// TIA Portal V19 export
FUNCTION "SUGAR TRANSFER CYCLE" : Void   // FC26, LAD
{ S7_Optimized_Access := 'TRUE' }
// stored: SetENOAutomatically false
   VAR_TEMP   // added for the SCL form of the ladder/FBD networks
      _w1 : Bool;
   END_VAR
BEGIN

REGION Network 1: TRANSFER SELECT
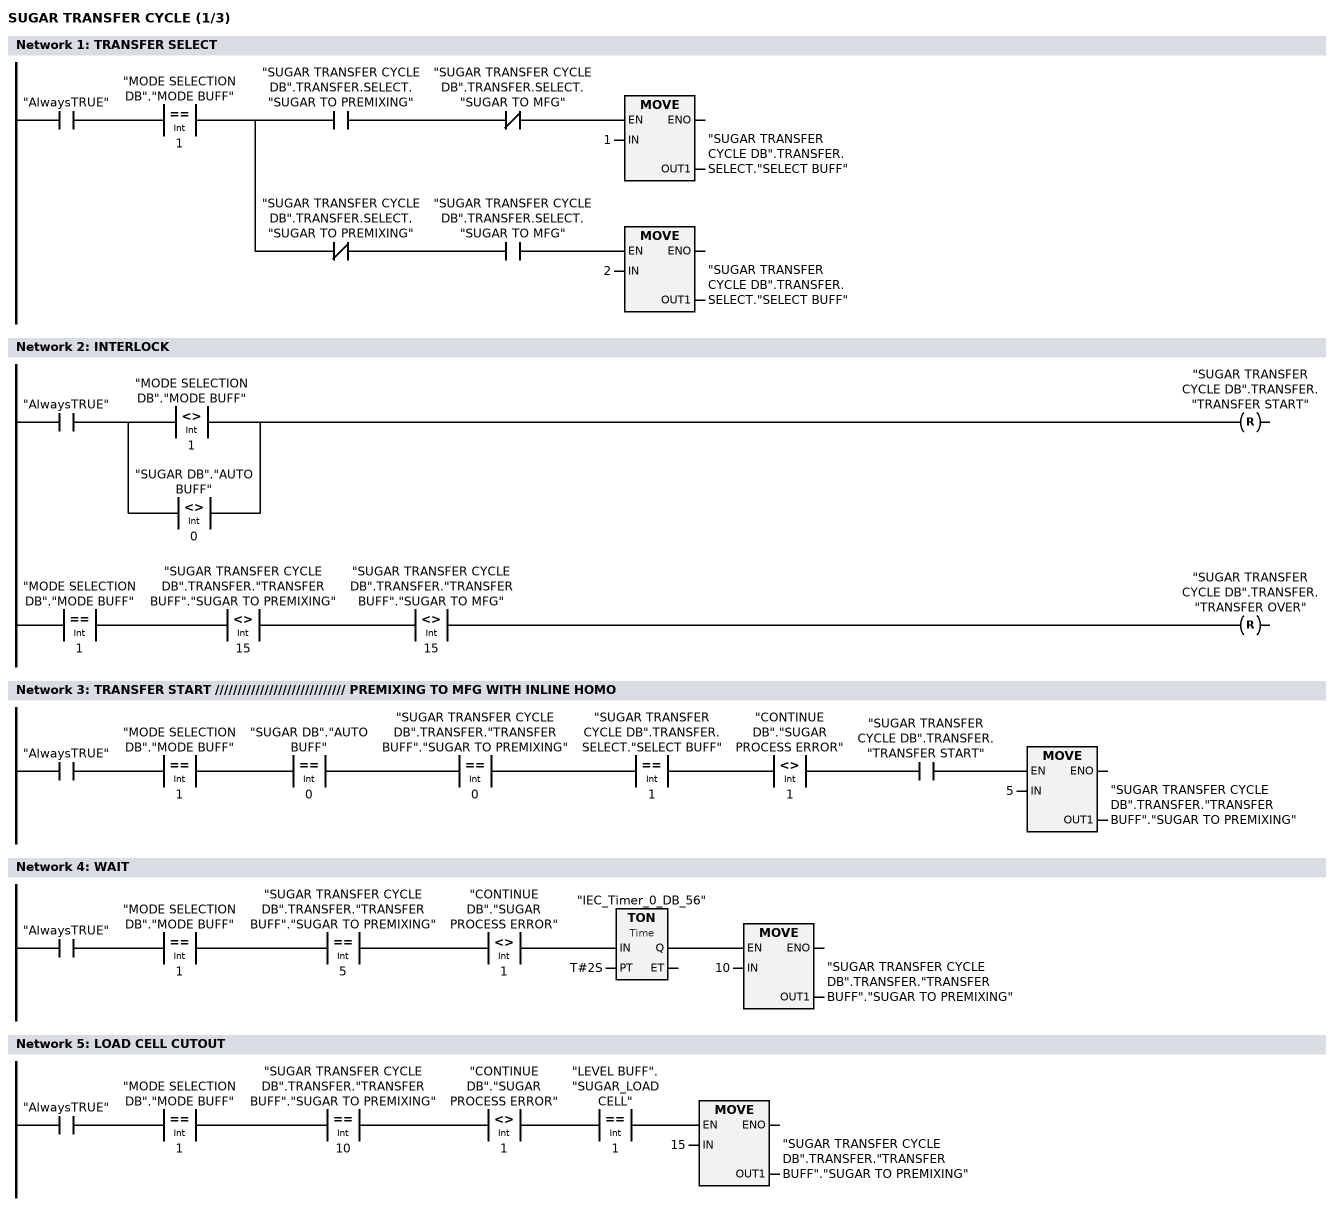
   RUNG wire#powerrail
      Contact( "AlwaysTRUE" )
      { S7_Templates := "SrcType := Int" } EQ_Contact(in1 := "MODE SELECTION DB"."MODE BUFF", in2 := 1)
      wire#w1
      Contact( "SUGAR TRANSFER CYCLE DB".TRANSFER.SELECT."SUGAR TO PREMIXING" )
      I_Contact( "SUGAR TRANSFER CYCLE DB".TRANSFER.SELECT."SUGAR TO MFG" )
      Move(in := 1, out1 => "SUGAR TRANSFER CYCLE DB".TRANSFER.SELECT."SELECT BUFF")
   END_RUNG
   RUNG wire#w1
      I_Contact( "SUGAR TRANSFER CYCLE DB".TRANSFER.SELECT."SUGAR TO PREMIXING" )
      Contact( "SUGAR TRANSFER CYCLE DB".TRANSFER.SELECT."SUGAR TO MFG" )
      Move(in := 2, out1 => "SUGAR TRANSFER CYCLE DB".TRANSFER.SELECT."SELECT BUFF")
   END_RUNG
   // the same network as SCL:
   #_w1 := "AlwaysTRUE" AND ("MODE SELECTION DB"."MODE BUFF" = 1);
   IF #_w1 AND "SUGAR TRANSFER CYCLE DB".TRANSFER.SELECT."SUGAR TO PREMIXING" AND NOT "SUGAR TRANSFER CYCLE DB".TRANSFER.SELECT."SUGAR TO MFG" THEN
       "SUGAR TRANSFER CYCLE DB".TRANSFER.SELECT."SELECT BUFF" := 1;
   END_IF;
   IF #_w1 AND NOT "SUGAR TRANSFER CYCLE DB".TRANSFER.SELECT."SUGAR TO PREMIXING" AND "SUGAR TRANSFER CYCLE DB".TRANSFER.SELECT."SUGAR TO MFG" THEN
       "SUGAR TRANSFER CYCLE DB".TRANSFER.SELECT."SELECT BUFF" := 2;
   END_IF;
END_REGION

REGION Network 2: INTERLOCK
   RUNG wire#powerrail
      Contact( "AlwaysTRUE" )
      wire#w1
      { S7_Templates := "SrcType := Int" } NE_Contact(in1 := "MODE SELECTION DB"."MODE BUFF", in2 := 1)
      wire#w2
      R_Coil( "SUGAR TRANSFER CYCLE DB".TRANSFER."TRANSFER START" )
   END_RUNG
   RUNG wire#w1
      { S7_Templates := "SrcType := Int" } NE_Contact(in1 := "SUGAR DB"."AUTO BUFF", in2 := 0)
   END_RUNG wire#w2
   RUNG wire#powerrail
      { S7_Templates := "SrcType := Int" } EQ_Contact(in1 := "MODE SELECTION DB"."MODE BUFF", in2 := 1)
      { S7_Templates := "SrcType := Int" } NE_Contact(in1 := "SUGAR TRANSFER CYCLE DB".TRANSFER."TRANSFER BUFF"."SUGAR TO PREMIXING", in2 := 15)
      { S7_Templates := "SrcType := Int" } NE_Contact(in1 := "SUGAR TRANSFER CYCLE DB".TRANSFER."TRANSFER BUFF"."SUGAR TO MFG", in2 := 15)
      R_Coil( "SUGAR TRANSFER CYCLE DB".TRANSFER."TRANSFER OVER" )
   END_RUNG
   // the same network as SCL:
   IF "AlwaysTRUE" AND (("MODE SELECTION DB"."MODE BUFF" <> 1) OR ("SUGAR DB"."AUTO BUFF" <> 0)) THEN
       "SUGAR TRANSFER CYCLE DB".TRANSFER."TRANSFER START" := FALSE;
   END_IF;
   IF ("MODE SELECTION DB"."MODE BUFF" = 1) AND ("SUGAR TRANSFER CYCLE DB".TRANSFER."TRANSFER BUFF"."SUGAR TO PREMIXING" <> 15) AND ("SUGAR TRANSFER CYCLE DB".TRANSFER."TRANSFER BUFF"."SUGAR TO MFG" <> 15) THEN
       "SUGAR TRANSFER CYCLE DB".TRANSFER."TRANSFER OVER" := FALSE;
   END_IF;
END_REGION

REGION Network 3: TRANSFER START ///////////////////////////// PREMIXING TO MFG WITH INLINE HOMO
   RUNG wire#powerrail
      Contact( "AlwaysTRUE" )
      { S7_Templates := "SrcType := Int" } EQ_Contact(in1 := "MODE SELECTION DB"."MODE BUFF", in2 := 1)
      { S7_Templates := "SrcType := Int" } EQ_Contact(in1 := "SUGAR DB"."AUTO BUFF", in2 := 0)
      { S7_Templates := "SrcType := Int" } EQ_Contact(in1 := "SUGAR TRANSFER CYCLE DB".TRANSFER."TRANSFER BUFF"."SUGAR TO PREMIXING", in2 := 0)
      { S7_Templates := "SrcType := Int" } EQ_Contact(in1 := "SUGAR TRANSFER CYCLE DB".TRANSFER.SELECT."SELECT BUFF", in2 := 1)
      { S7_Templates := "SrcType := Int" } NE_Contact(in1 := "CONTINUE DB"."SUGAR PROCESS ERROR", in2 := 1)
      Contact( "SUGAR TRANSFER CYCLE DB".TRANSFER."TRANSFER START" )
      Move(in := 5, out1 => "SUGAR TRANSFER CYCLE DB".TRANSFER."TRANSFER BUFF"."SUGAR TO PREMIXING")
   END_RUNG
   // the same network as SCL:
   IF "AlwaysTRUE" AND ("MODE SELECTION DB"."MODE BUFF" = 1) AND ("SUGAR DB"."AUTO BUFF" = 0) AND ("SUGAR TRANSFER CYCLE DB".TRANSFER."TRANSFER BUFF"."SUGAR TO PREMIXING" = 0) AND ("SUGAR TRANSFER CYCLE DB".TRANSFER.SELECT."SELECT BUFF" = 1) AND ("CONTINUE DB"."SUGAR PROCESS ERROR" <> 1) AND "SUGAR TRANSFER CYCLE DB".TRANSFER."TRANSFER START" THEN
       "SUGAR TRANSFER CYCLE DB".TRANSFER."TRANSFER BUFF"."SUGAR TO PREMIXING" := 5;
   END_IF;
END_REGION

REGION Network 4: WAIT
   RUNG wire#powerrail
      Contact( "AlwaysTRUE" )
      { S7_Templates := "SrcType := Int" } EQ_Contact(in1 := "MODE SELECTION DB"."MODE BUFF", in2 := 1)
      { S7_Templates := "SrcType := Int" } EQ_Contact(in1 := "SUGAR TRANSFER CYCLE DB".TRANSFER."TRANSFER BUFF"."SUGAR TO PREMIXING", in2 := 5)
      { S7_Templates := "SrcType := Int" } NE_Contact(in1 := "CONTINUE DB"."SUGAR PROCESS ERROR", in2 := 1)
      { S7_Templates := "time_type := Time" } "IEC_Timer_0_DB_56".TON(pt := T#2S, et =>)
      Move(in := 10, out1 => "SUGAR TRANSFER CYCLE DB".TRANSFER."TRANSFER BUFF"."SUGAR TO PREMIXING")
   END_RUNG
   // the same network as SCL:
   "IEC_Timer_0_DB_56".TON(IN := "AlwaysTRUE" AND ("MODE SELECTION DB"."MODE BUFF" = 1) AND ("SUGAR TRANSFER CYCLE DB".TRANSFER."TRANSFER BUFF"."SUGAR TO PREMIXING" = 5) AND ("CONTINUE DB"."SUGAR PROCESS ERROR" <> 1),
                           PT := T#2S);
   IF "IEC_Timer_0_DB_56".Q THEN
       "SUGAR TRANSFER CYCLE DB".TRANSFER."TRANSFER BUFF"."SUGAR TO PREMIXING" := 10;
   END_IF;
END_REGION

REGION Network 5: LOAD CELL CUTOUT
   RUNG wire#powerrail
      Contact( "AlwaysTRUE" )
      { S7_Templates := "SrcType := Int" } EQ_Contact(in1 := "MODE SELECTION DB"."MODE BUFF", in2 := 1)
      { S7_Templates := "SrcType := Int" } EQ_Contact(in1 := "SUGAR TRANSFER CYCLE DB".TRANSFER."TRANSFER BUFF"."SUGAR TO PREMIXING", in2 := 10)
      { S7_Templates := "SrcType := Int" } NE_Contact(in1 := "CONTINUE DB"."SUGAR PROCESS ERROR", in2 := 1)
      { S7_Templates := "SrcType := Int" } EQ_Contact(in1 := "LEVEL BUFF"."SUGAR_LOAD CELL", in2 := 1)
      Move(in := 15, out1 => "SUGAR TRANSFER CYCLE DB".TRANSFER."TRANSFER BUFF"."SUGAR TO PREMIXING")
   END_RUNG
   // the same network as SCL:
   IF "AlwaysTRUE" AND ("MODE SELECTION DB"."MODE BUFF" = 1) AND ("SUGAR TRANSFER CYCLE DB".TRANSFER."TRANSFER BUFF"."SUGAR TO PREMIXING" = 10) AND ("CONTINUE DB"."SUGAR PROCESS ERROR" <> 1) AND ("LEVEL BUFF"."SUGAR_LOAD CELL" = 1) THEN
       "SUGAR TRANSFER CYCLE DB".TRANSFER."TRANSFER BUFF"."SUGAR TO PREMIXING" := 15;
   END_IF;
END_REGION

REGION Network 6: TIMER
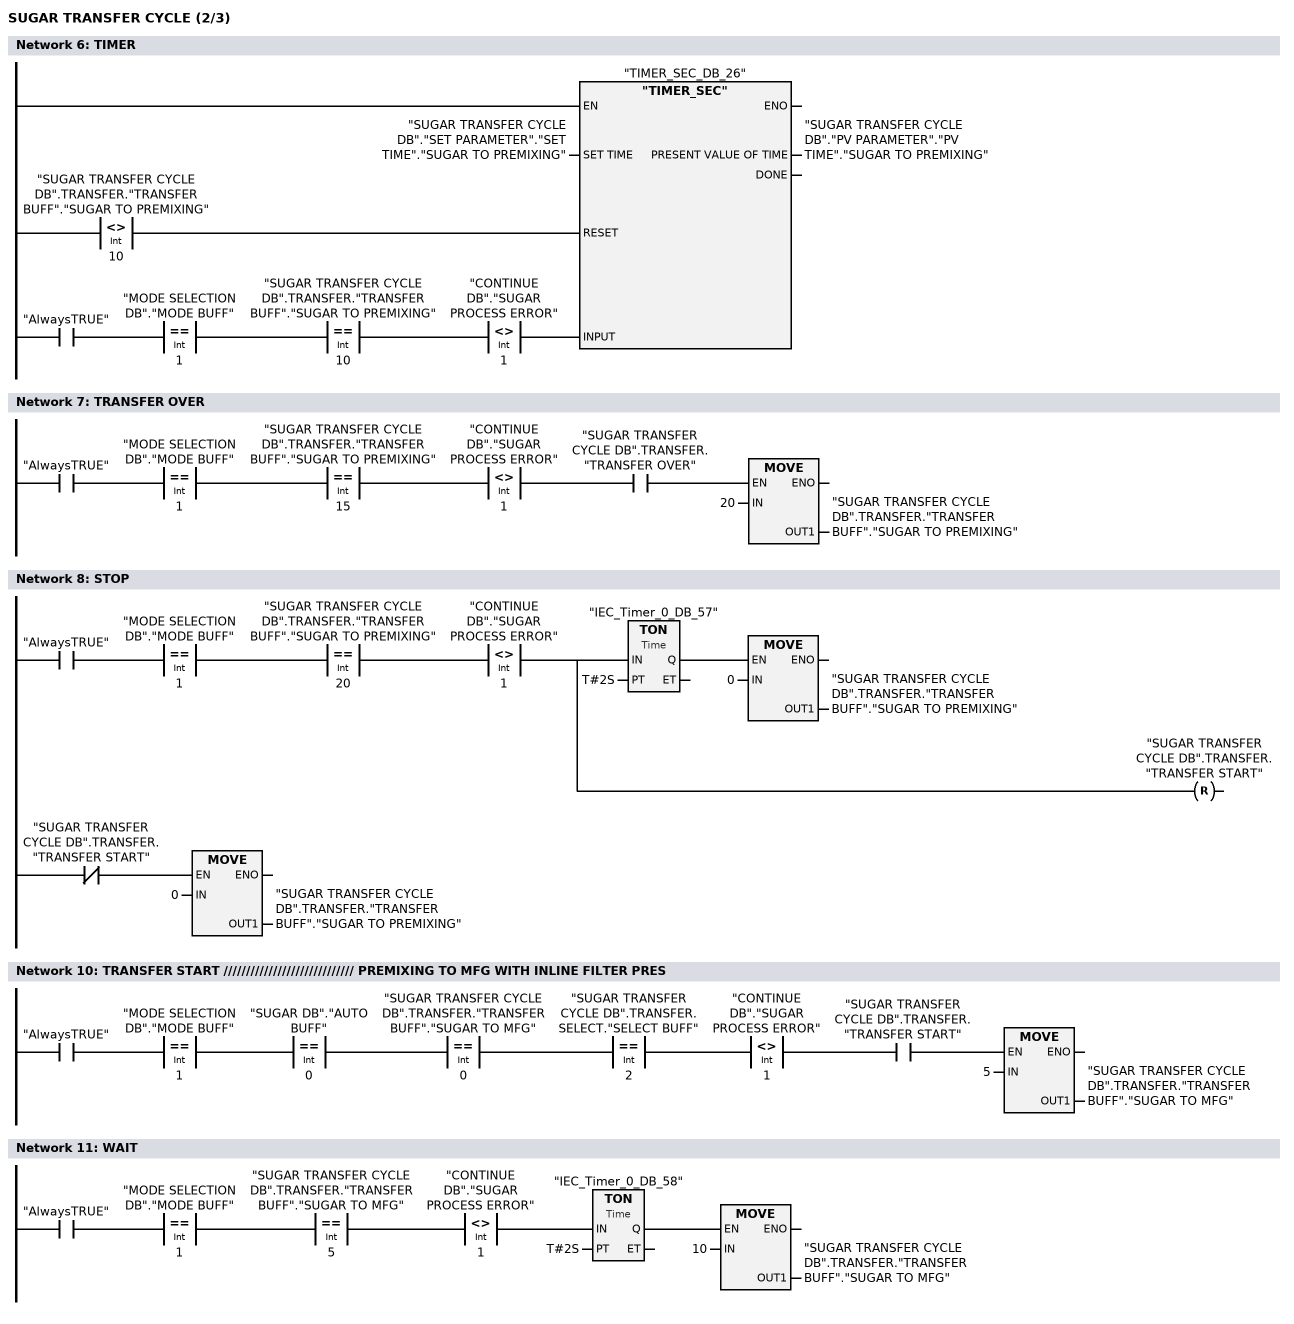
   RUNG wire#powerrail
      "TIMER_SEC_DB_26"(RESET := wire#w1, INPUT := wire#w2, "SET TIME" := "SUGAR TRANSFER CYCLE DB"."SET PARAMETER"."SET TIME"."SUGAR TO PREMIXING", "PRESENT VALUE OF TIME" => "SUGAR TRANSFER CYCLE DB"."PV PARAMETER"."PV TIME"."SUGAR TO PREMIXING", DONE =>)
   END_RUNG
   RUNG wire#powerrail
      { S7_Templates := "SrcType := Int" } NE_Contact(in1 := "SUGAR TRANSFER CYCLE DB".TRANSFER."TRANSFER BUFF"."SUGAR TO PREMIXING", in2 := 10)
   END_RUNG wire#w1
   RUNG wire#powerrail
      Contact( "AlwaysTRUE" )
      { S7_Templates := "SrcType := Int" } EQ_Contact(in1 := "MODE SELECTION DB"."MODE BUFF", in2 := 1)
      { S7_Templates := "SrcType := Int" } EQ_Contact(in1 := "SUGAR TRANSFER CYCLE DB".TRANSFER."TRANSFER BUFF"."SUGAR TO PREMIXING", in2 := 10)
      { S7_Templates := "SrcType := Int" } NE_Contact(in1 := "CONTINUE DB"."SUGAR PROCESS ERROR", in2 := 1)
   END_RUNG wire#w2
   // the same network as SCL:
   "TIMER_SEC_DB_26"("SET TIME" := "SUGAR TRANSFER CYCLE DB"."SET PARAMETER"."SET TIME"."SUGAR TO PREMIXING",   // "TIMER_SEC"
                     RESET := "SUGAR TRANSFER CYCLE DB".TRANSFER."TRANSFER BUFF"."SUGAR TO PREMIXING" <> 10,
                     INPUT := "AlwaysTRUE" AND ("MODE SELECTION DB"."MODE BUFF" = 1) AND ("SUGAR TRANSFER CYCLE DB".TRANSFER."TRANSFER BUFF"."SUGAR TO PREMIXING" = 10) AND ("CONTINUE DB"."SUGAR PROCESS ERROR" <> 1),
                     "PRESENT VALUE OF TIME" => "SUGAR TRANSFER CYCLE DB"."PV PARAMETER"."PV TIME"."SUGAR TO PREMIXING");
END_REGION

REGION Network 7: TRANSFER OVER
   RUNG wire#powerrail
      Contact( "AlwaysTRUE" )
      { S7_Templates := "SrcType := Int" } EQ_Contact(in1 := "MODE SELECTION DB"."MODE BUFF", in2 := 1)
      { S7_Templates := "SrcType := Int" } EQ_Contact(in1 := "SUGAR TRANSFER CYCLE DB".TRANSFER."TRANSFER BUFF"."SUGAR TO PREMIXING", in2 := 15)
      { S7_Templates := "SrcType := Int" } NE_Contact(in1 := "CONTINUE DB"."SUGAR PROCESS ERROR", in2 := 1)
      Contact( "SUGAR TRANSFER CYCLE DB".TRANSFER."TRANSFER OVER" )
      Move(in := 20, out1 => "SUGAR TRANSFER CYCLE DB".TRANSFER."TRANSFER BUFF"."SUGAR TO PREMIXING")
   END_RUNG
   // the same network as SCL:
   IF "AlwaysTRUE" AND ("MODE SELECTION DB"."MODE BUFF" = 1) AND ("SUGAR TRANSFER CYCLE DB".TRANSFER."TRANSFER BUFF"."SUGAR TO PREMIXING" = 15) AND ("CONTINUE DB"."SUGAR PROCESS ERROR" <> 1) AND "SUGAR TRANSFER CYCLE DB".TRANSFER."TRANSFER OVER" THEN
       "SUGAR TRANSFER CYCLE DB".TRANSFER."TRANSFER BUFF"."SUGAR TO PREMIXING" := 20;
   END_IF;
END_REGION

REGION Network 8: STOP
   RUNG wire#powerrail
      Contact( "AlwaysTRUE" )
      { S7_Templates := "SrcType := Int" } EQ_Contact(in1 := "MODE SELECTION DB"."MODE BUFF", in2 := 1)
      { S7_Templates := "SrcType := Int" } EQ_Contact(in1 := "SUGAR TRANSFER CYCLE DB".TRANSFER."TRANSFER BUFF"."SUGAR TO PREMIXING", in2 := 20)
      { S7_Templates := "SrcType := Int" } NE_Contact(in1 := "CONTINUE DB"."SUGAR PROCESS ERROR", in2 := 1)
      wire#w1
      { S7_Templates := "time_type := Time" } "IEC_Timer_0_DB_57".TON(pt := T#2S, et =>)
      Move(in := 0, out1 => "SUGAR TRANSFER CYCLE DB".TRANSFER."TRANSFER BUFF"."SUGAR TO PREMIXING")
   END_RUNG
   RUNG wire#w1
      R_Coil( "SUGAR TRANSFER CYCLE DB".TRANSFER."TRANSFER START" )
   END_RUNG
   RUNG wire#powerrail
      I_Contact( "SUGAR TRANSFER CYCLE DB".TRANSFER."TRANSFER START" )
      Move(in := 0, out1 => "SUGAR TRANSFER CYCLE DB".TRANSFER."TRANSFER BUFF"."SUGAR TO PREMIXING")
   END_RUNG
   // the same network as SCL:
   #_w1 := "AlwaysTRUE" AND ("MODE SELECTION DB"."MODE BUFF" = 1) AND ("SUGAR TRANSFER CYCLE DB".TRANSFER."TRANSFER BUFF"."SUGAR TO PREMIXING" = 20) AND ("CONTINUE DB"."SUGAR PROCESS ERROR" <> 1);
   "IEC_Timer_0_DB_57".TON(IN := #_w1, PT := T#2S);
   IF "IEC_Timer_0_DB_57".Q THEN
       "SUGAR TRANSFER CYCLE DB".TRANSFER."TRANSFER BUFF"."SUGAR TO PREMIXING" := 0;
   END_IF;
   IF #_w1 THEN "SUGAR TRANSFER CYCLE DB".TRANSFER."TRANSFER START" := FALSE; END_IF;
   IF NOT "SUGAR TRANSFER CYCLE DB".TRANSFER."TRANSFER START" THEN
       "SUGAR TRANSFER CYCLE DB".TRANSFER."TRANSFER BUFF"."SUGAR TO PREMIXING" := 0;
   END_IF;
END_REGION

REGION Network 10: TRANSFER START ///////////////////////////// PREMIXING TO MFG WITH INLINE FILTER PRES
   RUNG wire#powerrail
      Contact( "AlwaysTRUE" )
      { S7_Templates := "SrcType := Int" } EQ_Contact(in1 := "MODE SELECTION DB"."MODE BUFF", in2 := 1)
      { S7_Templates := "SrcType := Int" } EQ_Contact(in1 := "SUGAR DB"."AUTO BUFF", in2 := 0)
      { S7_Templates := "SrcType := Int" } EQ_Contact(in1 := "SUGAR TRANSFER CYCLE DB".TRANSFER."TRANSFER BUFF"."SUGAR TO MFG", in2 := 0)
      { S7_Templates := "SrcType := Int" } EQ_Contact(in1 := "SUGAR TRANSFER CYCLE DB".TRANSFER.SELECT."SELECT BUFF", in2 := 2)
      { S7_Templates := "SrcType := Int" } NE_Contact(in1 := "CONTINUE DB"."SUGAR PROCESS ERROR", in2 := 1)
      Contact( "SUGAR TRANSFER CYCLE DB".TRANSFER."TRANSFER START" )
      Move(in := 5, out1 => "SUGAR TRANSFER CYCLE DB".TRANSFER."TRANSFER BUFF"."SUGAR TO MFG")
   END_RUNG
   // the same network as SCL:
   IF "AlwaysTRUE" AND ("MODE SELECTION DB"."MODE BUFF" = 1) AND ("SUGAR DB"."AUTO BUFF" = 0) AND ("SUGAR TRANSFER CYCLE DB".TRANSFER."TRANSFER BUFF"."SUGAR TO MFG" = 0) AND ("SUGAR TRANSFER CYCLE DB".TRANSFER.SELECT."SELECT BUFF" = 2) AND ("CONTINUE DB"."SUGAR PROCESS ERROR" <> 1) AND "SUGAR TRANSFER CYCLE DB".TRANSFER."TRANSFER START" THEN
       "SUGAR TRANSFER CYCLE DB".TRANSFER."TRANSFER BUFF"."SUGAR TO MFG" := 5;
   END_IF;
END_REGION

REGION Network 11: WAIT
   RUNG wire#powerrail
      Contact( "AlwaysTRUE" )
      { S7_Templates := "SrcType := Int" } EQ_Contact(in1 := "MODE SELECTION DB"."MODE BUFF", in2 := 1)
      { S7_Templates := "SrcType := Int" } EQ_Contact(in1 := "SUGAR TRANSFER CYCLE DB".TRANSFER."TRANSFER BUFF"."SUGAR TO MFG", in2 := 5)
      { S7_Templates := "SrcType := Int" } NE_Contact(in1 := "CONTINUE DB"."SUGAR PROCESS ERROR", in2 := 1)
      { S7_Templates := "time_type := Time" } "IEC_Timer_0_DB_58".TON(pt := T#2S, et =>)
      Move(in := 10, out1 => "SUGAR TRANSFER CYCLE DB".TRANSFER."TRANSFER BUFF"."SUGAR TO MFG")
   END_RUNG
   // the same network as SCL:
   "IEC_Timer_0_DB_58".TON(IN := "AlwaysTRUE" AND ("MODE SELECTION DB"."MODE BUFF" = 1) AND ("SUGAR TRANSFER CYCLE DB".TRANSFER."TRANSFER BUFF"."SUGAR TO MFG" = 5) AND ("CONTINUE DB"."SUGAR PROCESS ERROR" <> 1),
                           PT := T#2S);
   IF "IEC_Timer_0_DB_58".Q THEN
       "SUGAR TRANSFER CYCLE DB".TRANSFER."TRANSFER BUFF"."SUGAR TO MFG" := 10;
   END_IF;
END_REGION

REGION Network 12: LOAD CELL CUTOUT
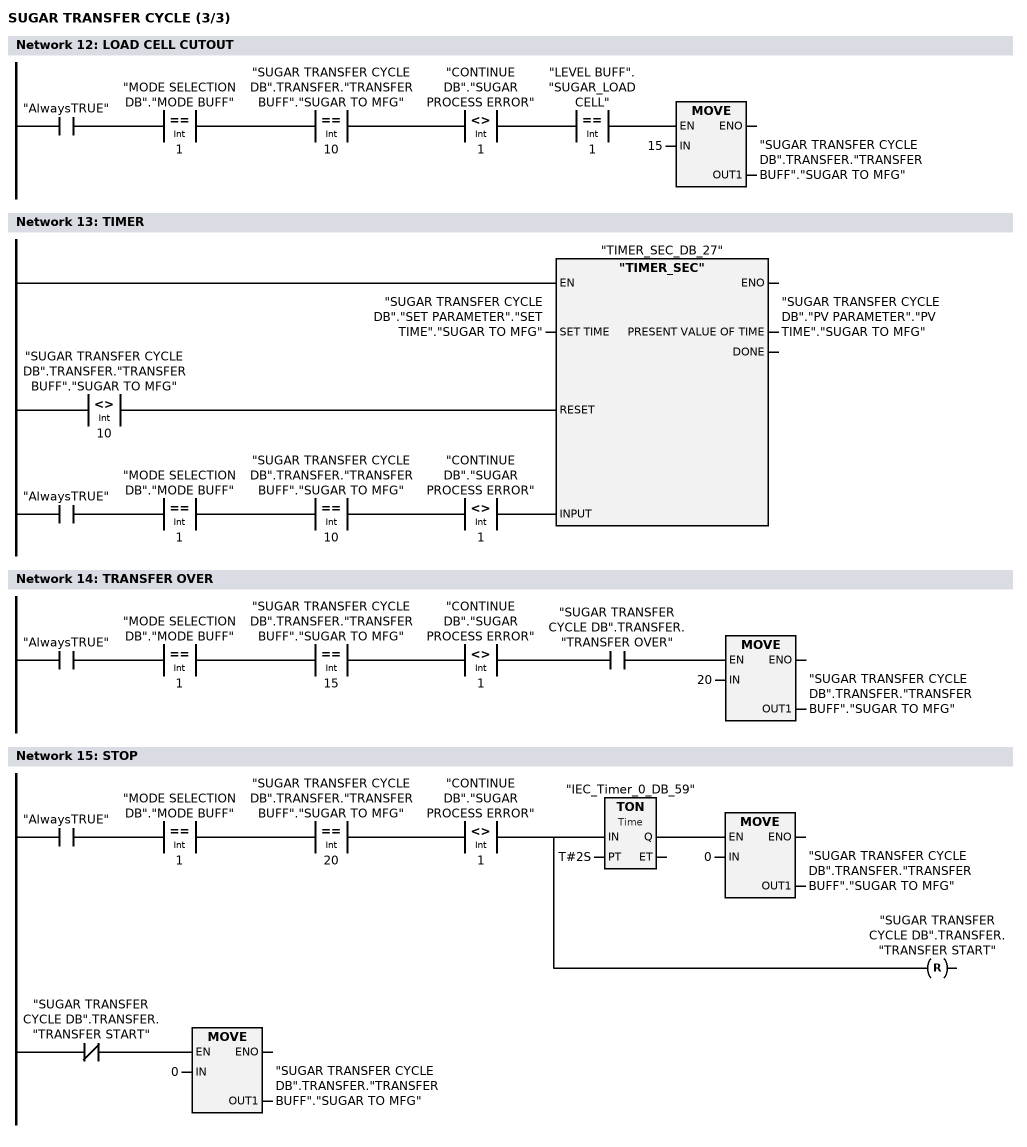
   RUNG wire#powerrail
      Contact( "AlwaysTRUE" )
      { S7_Templates := "SrcType := Int" } EQ_Contact(in1 := "MODE SELECTION DB"."MODE BUFF", in2 := 1)
      { S7_Templates := "SrcType := Int" } EQ_Contact(in1 := "SUGAR TRANSFER CYCLE DB".TRANSFER."TRANSFER BUFF"."SUGAR TO MFG", in2 := 10)
      { S7_Templates := "SrcType := Int" } NE_Contact(in1 := "CONTINUE DB"."SUGAR PROCESS ERROR", in2 := 1)
      { S7_Templates := "SrcType := Int" } EQ_Contact(in1 := "LEVEL BUFF"."SUGAR_LOAD CELL", in2 := 1)
      Move(in := 15, out1 => "SUGAR TRANSFER CYCLE DB".TRANSFER."TRANSFER BUFF"."SUGAR TO MFG")
   END_RUNG
   // the same network as SCL:
   IF "AlwaysTRUE" AND ("MODE SELECTION DB"."MODE BUFF" = 1) AND ("SUGAR TRANSFER CYCLE DB".TRANSFER."TRANSFER BUFF"."SUGAR TO MFG" = 10) AND ("CONTINUE DB"."SUGAR PROCESS ERROR" <> 1) AND ("LEVEL BUFF"."SUGAR_LOAD CELL" = 1) THEN
       "SUGAR TRANSFER CYCLE DB".TRANSFER."TRANSFER BUFF"."SUGAR TO MFG" := 15;
   END_IF;
END_REGION

REGION Network 13: TIMER
   RUNG wire#powerrail
      "TIMER_SEC_DB_27"(RESET := wire#w1, INPUT := wire#w2, "SET TIME" := "SUGAR TRANSFER CYCLE DB"."SET PARAMETER"."SET TIME"."SUGAR TO MFG", "PRESENT VALUE OF TIME" => "SUGAR TRANSFER CYCLE DB"."PV PARAMETER"."PV TIME"."SUGAR TO MFG", DONE =>)
   END_RUNG
   RUNG wire#powerrail
      { S7_Templates := "SrcType := Int" } NE_Contact(in1 := "SUGAR TRANSFER CYCLE DB".TRANSFER."TRANSFER BUFF"."SUGAR TO MFG", in2 := 10)
   END_RUNG wire#w1
   RUNG wire#powerrail
      Contact( "AlwaysTRUE" )
      { S7_Templates := "SrcType := Int" } EQ_Contact(in1 := "MODE SELECTION DB"."MODE BUFF", in2 := 1)
      { S7_Templates := "SrcType := Int" } EQ_Contact(in1 := "SUGAR TRANSFER CYCLE DB".TRANSFER."TRANSFER BUFF"."SUGAR TO MFG", in2 := 10)
      { S7_Templates := "SrcType := Int" } NE_Contact(in1 := "CONTINUE DB"."SUGAR PROCESS ERROR", in2 := 1)
   END_RUNG wire#w2
   // the same network as SCL:
   "TIMER_SEC_DB_27"("SET TIME" := "SUGAR TRANSFER CYCLE DB"."SET PARAMETER"."SET TIME"."SUGAR TO MFG",   // "TIMER_SEC"
                     RESET := "SUGAR TRANSFER CYCLE DB".TRANSFER."TRANSFER BUFF"."SUGAR TO MFG" <> 10,
                     INPUT := "AlwaysTRUE" AND ("MODE SELECTION DB"."MODE BUFF" = 1) AND ("SUGAR TRANSFER CYCLE DB".TRANSFER."TRANSFER BUFF"."SUGAR TO MFG" = 10) AND ("CONTINUE DB"."SUGAR PROCESS ERROR" <> 1),
                     "PRESENT VALUE OF TIME" => "SUGAR TRANSFER CYCLE DB"."PV PARAMETER"."PV TIME"."SUGAR TO MFG");
END_REGION

REGION Network 14: TRANSFER OVER
   RUNG wire#powerrail
      Contact( "AlwaysTRUE" )
      { S7_Templates := "SrcType := Int" } EQ_Contact(in1 := "MODE SELECTION DB"."MODE BUFF", in2 := 1)
      { S7_Templates := "SrcType := Int" } EQ_Contact(in1 := "SUGAR TRANSFER CYCLE DB".TRANSFER."TRANSFER BUFF"."SUGAR TO MFG", in2 := 15)
      { S7_Templates := "SrcType := Int" } NE_Contact(in1 := "CONTINUE DB"."SUGAR PROCESS ERROR", in2 := 1)
      Contact( "SUGAR TRANSFER CYCLE DB".TRANSFER."TRANSFER OVER" )
      Move(in := 20, out1 => "SUGAR TRANSFER CYCLE DB".TRANSFER."TRANSFER BUFF"."SUGAR TO MFG")
   END_RUNG
   // the same network as SCL:
   IF "AlwaysTRUE" AND ("MODE SELECTION DB"."MODE BUFF" = 1) AND ("SUGAR TRANSFER CYCLE DB".TRANSFER."TRANSFER BUFF"."SUGAR TO MFG" = 15) AND ("CONTINUE DB"."SUGAR PROCESS ERROR" <> 1) AND "SUGAR TRANSFER CYCLE DB".TRANSFER."TRANSFER OVER" THEN
       "SUGAR TRANSFER CYCLE DB".TRANSFER."TRANSFER BUFF"."SUGAR TO MFG" := 20;
   END_IF;
END_REGION

REGION Network 15: STOP
   RUNG wire#powerrail
      Contact( "AlwaysTRUE" )
      { S7_Templates := "SrcType := Int" } EQ_Contact(in1 := "MODE SELECTION DB"."MODE BUFF", in2 := 1)
      { S7_Templates := "SrcType := Int" } EQ_Contact(in1 := "SUGAR TRANSFER CYCLE DB".TRANSFER."TRANSFER BUFF"."SUGAR TO MFG", in2 := 20)
      { S7_Templates := "SrcType := Int" } NE_Contact(in1 := "CONTINUE DB"."SUGAR PROCESS ERROR", in2 := 1)
      wire#w1
      { S7_Templates := "time_type := Time" } "IEC_Timer_0_DB_59".TON(pt := T#2S, et =>)
      Move(in := 0, out1 => "SUGAR TRANSFER CYCLE DB".TRANSFER."TRANSFER BUFF"."SUGAR TO MFG")
   END_RUNG
   RUNG wire#w1
      R_Coil( "SUGAR TRANSFER CYCLE DB".TRANSFER."TRANSFER START" )
   END_RUNG
   RUNG wire#powerrail
      I_Contact( "SUGAR TRANSFER CYCLE DB".TRANSFER."TRANSFER START" )
      Move(in := 0, out1 => "SUGAR TRANSFER CYCLE DB".TRANSFER."TRANSFER BUFF"."SUGAR TO MFG")
   END_RUNG
   // the same network as SCL:
   #_w1 := "AlwaysTRUE" AND ("MODE SELECTION DB"."MODE BUFF" = 1) AND ("SUGAR TRANSFER CYCLE DB".TRANSFER."TRANSFER BUFF"."SUGAR TO MFG" = 20) AND ("CONTINUE DB"."SUGAR PROCESS ERROR" <> 1);
   "IEC_Timer_0_DB_59".TON(IN := #_w1, PT := T#2S);
   IF "IEC_Timer_0_DB_59".Q THEN
       "SUGAR TRANSFER CYCLE DB".TRANSFER."TRANSFER BUFF"."SUGAR TO MFG" := 0;
   END_IF;
   IF #_w1 THEN "SUGAR TRANSFER CYCLE DB".TRANSFER."TRANSFER START" := FALSE; END_IF;
   IF NOT "SUGAR TRANSFER CYCLE DB".TRANSFER."TRANSFER START" THEN
       "SUGAR TRANSFER CYCLE DB".TRANSFER."TRANSFER BUFF"."SUGAR TO MFG" := 0;
   END_IF;
END_REGION
END_FUNCTION
